//FUNCTION_BLOCK TcAxis_Tc2_MC2 EXTENDS TcAxis_Base IMPLEMENTS itfAxis_Tc2_MC2
//FUNCTION_BLOCK TcAxis_Tc2_MC2 EXTENDS TcAxis_DMC_Tc3_Direct_Motion_Control IMPLEMENTS itfAxis_Tc2_MC2
FUNCTION_BLOCK TcAxis_Tc2_MC2 IMPLEMENTS itfAxis_Tc2_MC2
//FUNCTION_BLOCK TcAxis_Tc2_MC2 EXTENDS TcAxis_Base IMPLEMENTS itfAxis_Tc3_DriveMotionControl, itfAxis_Tc2_MC2

//VAR_INPUT
//	Axis 				: Tc2_MC2.AXIS_REF;
//END_VAR
//VAR_OUTPUT
//END_VAR
VAR_IN_OUT 
	Axis 				: Tc2_MC2.AXIS_REF;
END_VAR
VAR	
	_PowerOn : BOOL;
//	itfCommand      : itfCommand;

//	_fbCommand       	: TcCommand;
	
	_fbAxisCommand   	: TcAxisCommand;

//itfAxisCommand  : itfAxisCommand;
//_Command         : ST_Command;
	

MC : ST_Tc2_MC2;	

count_delete : INT;	
END_VAR

 ACT_Cyclic_Update();

METHOD AbortTrigger : itfCommand
VAR_INPUT
END_VAR
END_METHOD

{warning 'add method implementation '}
METHOD AccelerationProfile 	: itfCommand
VAR_INPUT
	TimeScale				: REAL;
	AccelerationScale		: REAL;
	Offset					: REAL;
	BufferMode				: MC_BUFFER_MODE;
END_VAR
VAR
	
END_VAR
count_delete  := count_delete + 1;
END_METHOD

ACTION ACT_Cyclic_Update:
//update local variables from hardware
Axis.ReadStatus();
END_ACTION

{warning 'add property implementation'}
PROPERTY ActualPosition : REAL
GET
//Actual Position
IF Axis.Status.OpMode.Modulo THEN
    ActualPosition := Axis.NcToPlc.ModuloActPos;
ELSE
    ActualPosition := Axis.NcToPlc.ActPos;
END_IF

count_delete  := count_delete + 1;
END_GET
END_PROPERTY

{warning 'add property implementation'}
PROPERTY ActualTorque : REAL
GET
ActualTorque := Axis.NcToPlc.ActTorque;

count_delete  := count_delete + 1;
END_GET
END_PROPERTY

{warning 'add property implementation'}
PROPERTY ActualVelocity : REAL
GET
//Actual Velocity
ActualVelocity := Axis.NcToPlc.ActVelo;
END_GET
END_PROPERTY

{warning 'add property implementation'}
PROPERTY AxisWarning : BOOL
GET
count_delete  := count_delete + 1;
END_GET
END_PROPERTY

{warning 'add property implementation'}
PROPERTY CommunicationReady : BOOL
GET
count_delete  := count_delete + 1;
END_GET
END_PROPERTY

{warning 'add property implementation'}
PROPERTY Direction : AXIS_DIRECTION
GET
count_delete  := count_delete + 1;
END_GET
END_PROPERTY

PROPERTY Error : BOOL
GET
Error :=  Axis.Status.Error;
END_GET
END_PROPERTY

{warning 'add property implementation'}
PROPERTY ErrorId : WORD
GET

//ErrorId := Axis.Status.ErrorID;

count_delete  := count_delete + 1;
END_GET
END_PROPERTY

PROPERTY ErrorId_Udint_Status : UDINT
GET
ErrorId_Udint_Status := Axis.Status.ErrorID;
END_GET
END_PROPERTY

PROPERTY Geared : BOOL
GET
Geared :=  Axis.Status.Coupled;
//Axis.NcToPlc.CoupleState
END_GET
END_PROPERTY

{attribute 'TcRpcEnable'}
METHOD GearIn 			: itfSynchronizedAxisCommand
VAR_INPUT
	RatioNumerator		: LREAL;
	RatioDenominator	: UINT;
	Acceleration		: LREAL;
	Deceleration		: LREAL;
	Jerk				: LREAL;
//	BufferMode			: Tc2_MC2.MC_BufferMode; //Currently not implemented
//	Options             : Tc2_MC2.ST_GearInOptions; //Currently not implemented
END_VAR
VAR_IN_OUT 
	Slave				: Tc2_MC2.AXIS_REF;	
END_VAR
VAR
//	fbGearIn			: Tc2_MC2.MC_GearIn;	
END_VAR
	
MC.GearIn(
	Master:= Axis, 
	Slave:= Slave, 
	Execute:= TRUE, 
	RatioNumerator:= RatioNumerator, 
	RatioDenominator:= RatioDenominator, 
	Acceleration:= Acceleration,
	Deceleration:= Deceleration, 
	Jerk:= Jerk, 
	BufferMode:= , //BufferMode,
	Options:= , //Options, 
	InGear=> ,//Geared , 
	Busy=> , 
	Active=> , 
	CommandAborted=> , 
	Error=> , 
	ErrorID=> );
	
MC.GearIn(
	Master:= Axis, 
	Slave:= Slave, 
	Execute:= FALSE);
	
count_delete  := count_delete + 1;
END_METHOD

{attribute 'TcRpcEnable'}
METHOD GearInDyn 		: itfSynchronizedAxisCommand
VAR_INPUT
    GearRatio			: LREAL;
	Acceleration		: REAL;
	Deceleration		: REAL;
	Jerk				: REAL;
//	BufferMode			: Tc2_MC2.MC_BufferMode;
//	Options             : Tc2_MC2.ST_GearInDynOptions;
END_VAR

VAR_IN_OUT 
	Slave				: Tc2_MC2.AXIS_REF;	
END_VAR
END_METHOD

{attribute 'TcRpcEnable'}
METHOD GearInMultimaster 	: itfSynchronizedAxisCommand
VAR_INPUT
	GearRatio1				: LREAL;
	GearRatio2				: LREAL;
	GearRatio3				: LREAL;	
	GearRatio4				: LREAL;	
	Acceleration			: LREAL;
	Deceleration			: LREAL;
	Jerk					: LREAL;
	BufferMode				: Tc2_MC2.MC_BufferMode;
	Options             	: Tc2_MC2.ST_GearInMultiMasterOptions;	
END_VAR

VAR_IN_OUT
	Master1					: Tc2_MC2.AXIS_REF;	
	Master2					: Tc2_MC2.AXIS_REF;	
	Master3					: Tc2_MC2.AXIS_REF;	
	Master4					: Tc2_MC2.AXIS_REF;	
	Slave					: Tc2_MC2.AXIS_REF;	
END_VAR
END_METHOD

{attribute 'TcRpcEnable'}
METHOD GearOut 			: itfSynchronizedAxisCommand
VAR_INPUT
	Options             : Tc2_MC2.ST_GearInDynOptions;
END_VAR

VAR_IN_OUT 
	Slave				: Tc2_MC2.AXIS_REF;	
END_VAR
END_METHOD

{warning 'add method implementation '}
METHOD Halt 		: itfAxisCommand
VAR_INPUT
	Deceleration	: REAL;
	Jerk			: REAL;
	BufferMode		: MC_BUFFER_MODE;
END_VAR
VAR
//	fbHalt			: Tc2_MC2.MC_HALT;
END_VAR

MC.Halt(
	Axis:= Axis, 
	Execute:= , 
	Deceleration:= Deceleration, 
	Jerk:= Jerk, 
	BufferMode:= , //BufferMode, 
	Options:= , 
	Done=> , 
	Busy=> , 
	Active=> , 
	CommandAborted=> , 
	Error=> , 
	ErrorID=> );

count_delete  := count_delete + 1;
END_METHOD

{warning 'add method implementation '}
METHOD HaltSuperimposed : itfAxisCommand
VAR_INPUT
	Deceleration		: REAL;
	Jerk				: REAL;
END_VAR
VAR
	
END_VAR
count_delete  := count_delete + 1;
END_METHOD

{warning 'add method implementation '}
METHOD Home 		: itfAxisCommand
VAR_INPUT
	Position		: REAL;
	Velocity		: REAL;
	EndVelocity		: REAL;
	Acceleration	: REAL;
	Deceleration	: REAL;
	Jerk			: REAL;
	Direction		: MC_Direction;
	HomingMode		: INT;
	BufferMode		: MC_BUFFER_MODE;
END_VAR
VAR
//	fbHome			: Tc2_MC2.MC_HOME;
END_VAR

MC.Home(
	Axis:= Axis, 
	Execute:= TRUE, 
	Position:= Position, 
	HomingMode:= HomingMode, 
	BufferMode:= ,//BufferMode , 
	Options:= , 
	bCalibrationCam:= , 
	Done=> , 
	Busy=> , 
	Active=> , 
	CommandAborted=> , 
	Error=> , 
	ErrorID=> );

count_delete  := count_delete + 1;
END_METHOD

{warning 'add property implementation'}
PROPERTY HomeAbsSwitch : BOOL
GET
count_delete  := count_delete + 1;
END_GET
END_PROPERTY


PROPERTY IsHomed : BOOL
GET

IsHomed := Axis.Status.Homed;
END_GET
END_PROPERTY

{warning 'add method implementation '}
METHOD Jog 			: itfAxisCommand
VAR_INPUT
    JogForward 		: BOOL;
    JogBackwards 	: BOOL;
    Mode     		: Tc2_MC2.E_JogMode;
    Position        : LREAL;
    Velocity        : LREAL;
    Acceleration 	: LREAL;
    Deceleration 	: LREAL;
    Jerk     		: LREAL;
END_VAR
VAR
//	fbJog			: Tc2_MC2.MC_JOG;
END_VAR

MC.Jog(
	Axis:= Axis, 
	JogForward:= JogForward, 
	JogBackwards:= JogBackwards, 
	Mode:= Mode, 
	Position:= Position, 
	Velocity:= Velocity, 
	Acceleration:= Acceleration, 
	Deceleration:= Deceleration, 
	Jerk:= Jerk, 
	Done=> , 
	Busy=> , 
	Active=> , 
	CommandAborted=> , 
	Error=> , 
	ErrorID=> );


count_delete  := count_delete + 1;
END_METHOD

{warning 'add property implementation'}
PROPERTY LimitSwitchNegative : BOOL
GET

LimitSwitchNegative := Axis.Status.SoftLimitMinExceeded;

count_delete  := count_delete + 1;
END_GET
END_PROPERTY

{warning 'add property implementation'}
PROPERTY LimitSwitchPositive : BOOL
GET

LimitSwitchPositive := Axis.Status.SoftLimitMaxExceeded;

count_delete  := count_delete + 1;
END_GET
END_PROPERTY

{warning 'add property implementation'}
PROPERTY MotionStatus : MOTION_STATUS
GET
END_GET
END_PROPERTY

{attribute 'TcRpcEnable'}
METHOD MoveAbsolute : itfAxisCommand
VAR_INPUT
	Position		: REAL;
	Velocity		: REAL;
	Acceleration	: REAL;
	Deceleration	: REAL;
	Jerk			: REAL;
//	Direction		: MC_Direction;
	BufferMode		: MC_BUFFER_MODE;
//	Options         : Tc2_MC2.ST_MoveOptions;
	Options         : Tc2_Mc2.ST_MoveOptions;
END_VAR

VAR
	itfAxisCommand   : itfAxisCommand;
    _Command         : ST_Command;
END_VAR
itfAxisCommand := _fbAxisCommand;
	
MC.MoveAbsolute(
	Axis:= Axis, 
	Execute:= TRUE ,//Execute, //
	Position:= Position, 
	Velocity:= Velocity, 
	Acceleration:= Acceleration, 
	Deceleration:= Deceleration, 
	Jerk:= Jerk, 
	BufferMode:= BufferMode,//BufferMode, 
	Options:= Options, //Options, 
	Done=> _Command.Done, 
	Busy=> _Command.Busy, 
	Active=>_Command.Active, 
	CommandAborted=> _Command.CommandAborted, 
	Error=> _Command.Error, 
	ErrorID=> _Command.ErrorID_Udint);
	
MC.MoveAbsolute(
	Axis:= Axis, 
	Execute:= FALSE);	

itfAxisCommand.Done 				:=  _Command.Done AND ActualPosition = Position;             
itfAxisCommand.Busy   				:=	_Command.Busy;
itfAxisCommand.Active 				:=	_Command.Active;
itfAxisCommand.CommandAborted		:=	_Command.CommandAborted;
itfAxisCommand.Error 				:=	_Command.Error;
itfAxisCommand.ErrorID_Udint 		:=	_Command.ErrorID_Udint;

MoveAbsolute := itfAxisCommand;
END_METHOD

{warning 'add method implementation '}
METHOD MoveAdditive : itfAxisCommand
VAR_INPUT
	Distance		: REAL;
	Velocity		: REAL;
	Acceleration	: REAL;
	Deceleration	: REAL;
	Jerk			: REAL;
	BufferMode		: MC_BUFFER_MODE;
END_VAR
VAR
//	fbMoveAdditive 	: Tc2_MC2.MC_MoveAdditive;	
END_VAR

MC.MoveAdditive(
	Axis:= Axis, 
	Execute:= TRUE, 
	Distance:= Distance, 
	Velocity:= Velocity, 
	Acceleration:= Acceleration, 
	Deceleration:= Deceleration, 
	Jerk:= Jerk, 
	BufferMode:= , //BufferMode, 
	Options:= , 
	Done=> , 
	Busy=> , 
	Active=> , 
	CommandAborted=> , 
	Error=> , 
	ErrorID=> );


count_delete  := count_delete + 1;
END_METHOD

{warning 'add method implementation '}
METHOD MoveContinuousAbsolute 	: itfContinuousAxisCommand
VAR_INPUT
	Position					: REAL;
	EndVelocity					: REAL;
	Velocity					: REAL;
	Acceleration				: REAL;
	Deceleration				: REAL;
	Jerk						: REAL;
	Direction					: MC_DIRECTION;
	BufferMode					: MC_BUFFER_MODE;
END_VAR
VAR
//	fbMoveContinuousAbsolute 	: Tc2_MC2.MC_MoveContinuousAbsolute;		
END_VAR

MC.MoveContinuousAbsolute(
	Axis:= Axis, 
	Execute:= TRUE, 
	Position:= Position, 
	Velocity:= Velocity, 
	EndVelocity:= EndVelocity, 
	Acceleration:= Acceleration, 
	Deceleration:= Deceleration, 
	Jerk:= Jerk, 
	BufferMode:= ,//BufferMode, 
	Options:= , 
	InEndVelocity=> , 
	Busy=> , 
	Active=> , 
	CommandAborted=> , 
	Error=> , 
	ErrorID=> );


count_delete  := count_delete + 1;
END_METHOD

{warning 'add method implementation '}
METHOD MoveContinuousRelative 	: itfContinuousAxisCommand
VAR_INPUT
	Distance					: REAL;
	EndVelocity					: REAL;
	Velocity					: REAL;
	Acceleration				: REAL;
	Deceleration				: REAL;
	Jerk						: REAL;
	Direction					: MC_DIRECTION;
	BufferMode					: MC_BUFFER_MODE;
END_VAR
VAR
//	fbMoveContinuousRelative 	: Tc2_MC2.MC_MoveContinuousRelative;
END_VAR

MC.MoveContinuousRelative(
	Axis:= Axis, 
	Execute:= TRUE, 
	Distance:= Distance, 
	Velocity:= Velocity, 
	EndVelocity:= EndVelocity, 
	Acceleration:= Acceleration, 
	Deceleration:= Deceleration, 
	Jerk:= Jerk, 
	BufferMode:= ,//BufferMode, 
	Options:= , 
	InEndVelocity=> , 
	Busy=> , 
	Active=> , 
	CommandAborted=> , 
	Error=> , 
	ErrorID=> );



count_delete  := count_delete + 1;
END_METHOD

METHOD MoveModulo : itfAxisCommand
VAR_INPUT
END_VAR

MC.MoveModulo(
	Axis:= Axis, 
	Execute:= TRUE, 
	Position:= , 
	Velocity:= , 
	Acceleration:= , 
	Deceleration:= , 
	Jerk:= , 
	Direction:= , 
	BufferMode:= , 
	Options:= , 
	Done=> , 
	Busy=> , 
	Active=> , 
	CommandAborted=> , 
	Error=> , 
	ErrorID=> );
END_METHOD

{attribute 'TcRpcEnable'}
METHOD MoveRelative 	: itfAxisCommand
VAR_INPUT
	Distance			: REAL;
	Velocity			: REAL;
	Acceleration		: REAL;
	Deceleration		: REAL;
	Jerk				: REAL;
	BufferMode			: MC_BUFFER_MODE;
	Options         	: TC2_MC2.ST_MoveOptions;
END_VAR
VAR
	itfAxisCommand   : itfAxisCommand;
	_Command         : ST_Command;
END_VAR
itfAxisCommand := _fbAxisCommand;

MC.MoveRelative(
	Axis:= Axis, 
	Execute:= TRUE, 
	Distance:= Distance, 
	Velocity:= Velocity, 
	Acceleration:= Acceleration, 
	Deceleration:= Deceleration, 
	Jerk:= Jerk, 
	BufferMode:= ,//BufferMode, 
	Options:= Options, 
	Done=> _Command.Done, 
	Busy=> _Command.Busy, 
	Active=> _Command.Active, 
	CommandAborted=> _Command.CommandAborted, 
	Error=> _Command.Error, 
	ErrorID=> _Command.ErrorID_Udint);
	
MC.MoveRelative(
	Axis:= Axis, 
	Execute:= FALSE);		
	
itfAxisCommand.Done 				:=  _Command.Done; //AND ActualPosition = ActualPosition + Distance;             
itfAxisCommand.Busy   				:=	_Command.Busy;
itfAxisCommand.Active 				:=	_Command.Active;
itfAxisCommand.CommandAborted		:=	_Command.CommandAborted;
itfAxisCommand.Error 				:=	_Command.Error;
itfAxisCommand.ErrorID_Udint 		:=	_Command.ErrorID_Udint;

MoveRelative := itfAxisCommand;
END_METHOD

{warning 'add method implementation '}
METHOD MoveSuperimposed 	: itfAxisCommand
VAR_INPUT
	Distance				: REAL;
	VelocityDiff			: REAL;
	Acceleration			: REAL;
	Deceleration			: REAL;
	Jerk					: REAL;
END_VAR
VAR
//	fbMoveSuperimposed	 	: Tc2_MC2.MC_MoveSuperimposed;	
END_VAR

MC.MoveSuperimposed(
	Axis:= Axis, 
	Execute:= TRUE, 
	Mode:= , 
	Distance:= , 
	VelocityDiff:= VelocityDiff, 
	Acceleration:= Acceleration, 
	Deceleration:= Deceleration, 
	Jerk:= Jerk, 
	VelocityProcess:= , 
	Length:= , 
	Options:= , 
	Done=> , 
	Busy=> , 
	Active=> , 
	CommandAborted=> , 
	Error=> , 
	ErrorID=> , 
	Warning=> , 
	WarningId=> , 
	ActualVelocityDiff=> , 
	ActualDistance=> , 
	ActualLength=> , 
	ActualAcceleration=> , 
	ActualDeceleration=> );

count_delete  := count_delete + 1;
END_METHOD

{warning 'add method implementation '}
METHOD MoveVelocity 	: itfContinuousAxisCommand
VAR_INPUT
	Velocity			: REAL;
	Acceleration		: REAL;
	Deceleration		: REAL;
	Jerk				: REAL;
	Direction			: MC_Direction;
	BufferMode			: MC_BUFFER_MODE;
END_VAR
VAR
//	fbMoveVelocity	 	: Tc2_MC2.MC_MoveVelocity;	
END_VAR

MC.MoveVelocity(
	Axis:= Axis, 
	Execute:= TRUE, 
	Velocity:= Velocity, 
	Acceleration:= Acceleration, 
	Deceleration:= Deceleration, 
	Jerk:= Jerk, 
	Direction:= Direction, 
	BufferMode:= , //BufferMode
	Options:= , 
	InVelocity=> , 
	Busy=> , 
	Active=> , 
	CommandAborted=> , 
	Error=> , 
	ErrorID=> );	

count_delete  := count_delete + 1;
END_METHOD

{warning 'add method implementation '}
METHOD PhasingAbsolute 	: itfSynchronizedAxisCommand
VAR_INPUT
//	Master				: itfAxis;
	Master				: Tc2_MC2.AXIS_REF;
	Slave				: Tc2_MC2.AXIS_REF;		
	PhaseShift			: REAL;
	Velocity			: REAL;
	Acceleration		: REAL;
	Deceleration		: REAL;
	Jerk				: REAL;
	BufferMode			: MC_BUFFER_MODE;
END_VAR
VAR
//	fbPhasingAbsolute	: Tc2_MC2.MC_PhasingAbsolute;
END_VAR

MC.PhasingAbsolute(
	Master:= Master, 
	Slave:= Slave, 
	Execute:= TRUE, 
	ContinuousUpdate:= , 
	PhaseShift:= , 
	Velocity:= , 
	Acceleration:= , 
	Deceleration:= , 
	Jerk:= , 
	BufferMode:= , 
	Options:= , 
	Done=> , 
	Busy=> , 
	Active=> , 
	CommandAborted=> , 
	Error=> , 
	ErrorID=> , 
	AbsolutePhaseShift=> );

count_delete  := count_delete + 1;
END_METHOD

{warning 'add method implementation '}
METHOD PhasingRelative 	: itfSynchronizedAxisCommand
VAR_INPUT
//	Master				: itfAxis;
	Master				: Tc2_MC2.AXIS_REF;
	Slave				: Tc2_MC2.AXIS_REF;		
	PhaseShift			: REAL;
	Velocity			: REAL;
	Acceleration		: REAL;
	Deceleration		: REAL;
	Jerk				: REAL;
	BufferMode			: MC_BUFFER_MODE;
END_VAR
VAR
//	fbPhasingRelative	: Tc2_MC2.MC_PhasingRelative;
END_VAR

MC.PhasingRelative(
	Master:= Master, 
	Slave:= Slave, 
	Execute:= , 
	ContinuousUpdate:= , 
	PhaseShift:= , 
	Velocity:= , 
	Acceleration:= , 
	Deceleration:= , 
	Jerk:= , 
	BufferMode:= , 
	Options:= , 
	Done=> , 
	Busy=> , 
	Active=> , 
	CommandAborted=> , 
	Error=> , 
	ErrorID=> , 
	CoveredPhaseShift=> );

count_delete  := count_delete + 1;
END_METHOD

{warning 'add method implementation '}
METHOD PositionProfile 	: itfCommand
VAR_INPUT
	TimeScale			: REAL;
	PositionScale		: REAL;
	Offset				: REAL;
	BufferMode			: MC_BUFFER_MODE;
END_VAR
VAR
//	fbPositionProfile	 	: Tc2_MC2.;	
END_VAR






count_delete  := count_delete + 1;
END_METHOD

{attribute 'TcRpcEnable'}
METHOD Power 		: itfCommand
VAR_INPUT
	Enable			: BOOL;
	EnablePositive	: BOOL;
	EnableNegative	: BOOL;
END_VAR
VAR
	_fbCommand      : TcCommand;
	itfCommand      : itfCommand;
	Command         : ST_Command;
END_VAR

itfCommand := _fbCommand;

MC.Power(
	Axis:= Axis, 
	Enable:= Enable, 
	Enable_Positive:= EnablePositive, 
	Enable_Negative:= EnableNegative, 
	Override:= 100, 
	BufferMode:= , 
	Options:= , 
	Status=> Command.Status, 
	Busy=> Command.Busy,
	Active=> Command.Active,
	Error=> Command.Error,
	ErrorID=> Command.ErrorID_Udint);

itfCommand.Status		:=	Command.Status;
itfCommand.Busy   		:=	Command.Busy;
itfCommand.Active 		:=	Command.Active;
itfCommand.Error 		:=	Command.Error;
itfCommand.ErrorID_Udint :=	Command.ErrorID_Udint;
	
Power := itfCommand;

_PowerOn := MC.Power.Enable;
END_METHOD

{attribute ‘monitoring’ := ‘call’}
PROPERTY PowerOn : BOOL
GET
PowerOn := _PowerOn;
END_GET
END_PROPERTY

{warning 'add method implementation '}
METHOD ReadBoolParameter 	: MC_Error
VAR_INPUT
	ParameterNumber			: INT;
END_VAR
VAR_OUTPUT
	Value					: BOOL;
END_VAR
VAR
//	fbReadBoolParameter 	: Tc2_MC2.MC_ReadBoolParameter;
END_VAR

MC.ReadBoolParameter(
	Axis:= Axis, 
	Enable:= TRUE, 
	ParameterNumber:= ParameterNumber, 
	ReadMode:= , 
	Valid=> , 
	Busy=> , 
	Error=> , 
	ErrorID=> , 
	Value=> Value);


count_delete  := count_delete + 1;
END_METHOD

{warning 'add method implementation '}
METHOD ReadParameter 	: MC_Error
VAR_INPUT
	ParameterNumber		: INT;
END_VAR
VAR_OUTPUT
	Value				: REAL;
END_VAR
VAR
//	fbReadParameter		: Tc2_MC2.MC_ReadParameter;
END_VAR

MC.ReadParameter(
	Axis:= Axis, 
	Enable:= TRUE, 
	ParameterNumber:= ParameterNumber, 
	ReadMode:= , 
	Valid=> , 
	Busy=> , 
	Error=> , 
	ErrorID=> , 
	Value=> Value);


count_delete  := count_delete + 1;
END_METHOD

{warning 'add property implementation'}
PROPERTY ReadyForPowerOn : BOOL
GET
count_delete  := count_delete + 1;
END_GET
END_PROPERTY

{warning 'add method implementation '}
METHOD Release : MC_Error

VAR
	
END_VAR
count_delete  := count_delete + 1;
END_METHOD

{attribute 'TcRpcEnable'}
METHOD Reset 		: itfCommand

VAR
//	fbReset 		: Tc2_MC2.MC_RESET;
END_VAR

MC.Reset(
	Axis:= Axis, 
	Execute:= TRUE, 
	Done=> , 
	Busy=> , 
	Error=> , 
	ErrorID=> );


count_delete  := count_delete + 1;
END_METHOD

{warning 'add method implementation '}
METHOD SetOverride 	: MC_Error
VAR_INPUT
	VelFactor		: REAL;
	AccFactor		: REAL;
	JerkFactor		: REAL;
END_VAR

VAR
//	fbSetOverride 	: Tc2_MC2.MC_SetOverride;
END_VAR

MC.SetOverride(
	Axis:= Axis, 
	Enable:= TRUE, 
	VelFactor:= VelFactor, 
	AccFactor:= AccFactor, 
	JerkFactor:= JerkFactor, 
	Enabled=> , 
	Busy=> , 
	Error=> , 
	ErrorID=> );

count_delete  := count_delete + 1;
END_METHOD

{warning 'add method implementation '}
METHOD SetPosition 	: itfCommand
VAR_INPUT
	Position		: REAL;
	Relative		: BOOL; (* RELATIVE=True, ABSOLUTE=False (Default)*)
//	ExecutionMode	: MC_ExecutionMode;
    ExecutionMode	: Tc2_MC2.ST_SetPositionOptions;
END_VAR

VAR
//	fbSetPosition 	: Tc2_MC2.MC_SetPosition;
END_VAR

MC.SetPosition(
	Axis:= Axis, 
	Execute:= TRUE, 
	Position:= Position, 
	Mode:= Relative, 
	Options:= ExecutionMode, 
	Done=> , 
	Busy=> , 
	Error=> , 
	ErrorID=> );

count_delete  := count_delete + 1;
END_METHOD

{warning 'add property implementation'}
PROPERTY Simulation : BOOL
GET
count_delete  := count_delete + 1;
END_GET
END_PROPERTY

{attribute ‘monitoring’ := ‘call’}
PROPERTY Status : Tc2_MC2.MC_AxisStates
GET
VAR	
	AxisStates : Tc2_MC2.MC_AxisStates;
END_VAR

//CASE Axis.Status.MotionState OF 
//     MC_AXISSTATE_UNDEFINED : 
//         AxisStates := MC_AxisStates.MC_AXISSTATE_UNDEFINED;
//	MC_AXISSTATE_DISABLED:
//		AxisStates := MC_AxisStates.MC_AXISSTATE_DISABLED;
//	MC_AXISSTATE_STANDSTILL:
//		AxisStates := MC_AxisStates.MC_AXISSTATE_STANDSTILL;
//	MC_AXISSTATE_ERRORSTOP:		
//		AxisStates := MC_AxisStates.MC_AXISSTATE_ERRORSTOP;
//	MC_AXISSTATE_STOPPING:			
//		AxisStates := MC_AxisStates.MC_AXISSTATE_STOPPING;
//	MC_AXISSTATE_HOMING:			
//		AxisStates := MC_AxisStates.MC_AXISSTATE_HOMING;
//	MC_AXISSTATE_DISCRETEMOTION:			
//		AxisStates := MC_AxisStates.MC_AXISSTATE_DISCRETEMOTION;
//	MC_AXISSTATE_CONTINOUSMOTION:			
//		AxisStates := MC_AxisStates.MC_AXISSTATE_CONTINOUSMOTION;
//	MC_AXISSTATE_SYNCHRONIZEDMOTION:			
//		AxisStates := MC_AxisStates.MC_AXISSTATE_SYNCHRONIZEDMOTION;
//END_CASE;

//Status := AxisStates;

Status := Axis.Status.MotionState;
END_GET
END_PROPERTY

{warning 'add method implementation '}
METHOD Stop 		: itfAxisCommand
VAR_INPUT
	Deceleration	: REAL;
	Jerk			: REAL;
END_VAR
VAR
//	fbStop			: Tc2_MC2.MC_STOP;
END_VAR

MC.Stop(
	Axis:= Axis, 
	Execute:= TRUE, 
	Deceleration:= Deceleration, 
	Jerk:= Jerk, 
	Options:= , 
	Done=> , 
	Busy=> , 
	Active=> , 
	CommandAborted=> , 
	Error=> , 
	ErrorID=> );

count_delete  := count_delete + 1;
END_METHOD

{warning 'add method implementation '}
METHOD TorqueControl 	: itfAxisCommand
VAR_INPUT
	Torque				: REAL;
	TorqueRamp			: REAL;
	Velocity			: REAL;
	Acceleration		: REAL;
	Deceleration		: REAL;
	Jerk				: REAL;
	Direction			: MC_DIRECTION;
	BufferMode			: MC_BUFFER_MODE;
END_VAR
VAR
//	fbTorqueControl		: Tc2_MC2.MC_TorqueControl;
END_VAR

MC.TorqueControl(
	Axis:= Axis, 
	Execute:= , 
	ContinuousUpdate:= , 
	Relative:= , 
	Torque:= Torque, 
	TorqueRamp:= TorqueRamp, 
	VelocityLimitHigh:= , 
	VelocityLimitLow:= , 
	BufferMode:= , 
	Options:= , 
	InTorque=> , 
	Busy=> , 
	Active=> , 
	CommandAborted=> , 
	Error=> , 
	ErrorId=> );

count_delete  := count_delete + 1;
END_METHOD

METHOD TouchProbe : itfCommand
VAR_INPUT
END_VAR
END_METHOD

{warning 'add method implementation '}
METHOD VelocityProfile 	: itfCommand
VAR_INPUT
	TimeScale			: REAL;
	VelocityScale		: REAL;
	Offset				: REAL;
	BufferMode			: MC_BUFFER_MODE;
END_VAR
VAR
	
END_VAR
count_delete  := count_delete + 1;
END_METHOD

{warning 'add method implementation '}
METHOD WriteBoolParameter 	: MC_Error
VAR_INPUT
	ParameterNumber			: INT;
	Value					: BOOL;
END_VAR

VAR
//	fbWriteBoolParameter 	: Tc2_MC2.MC_WriteBoolParameter;	
END_VAR

MC.WriteBoolParameter(
	Axis:= Axis, 
	Execute:= TRUE, 
	ParameterNumber:= ParameterNumber, 
	Value:= Value, 
	Done=> , 
	Busy=> , 
	Error=> , 
	ErrorID=> );

count_delete  := count_delete + 1;
END_METHOD

{warning 'add method implementation '}
METHOD WriteParameter 	: MC_Error
VAR_INPUT
	ParameterNumber		: INT;
	Value				: REAL;
END_VAR

VAR
//	fbWriteParameter 	: Tc2_MC2.MC_WriteParameter;	
END_VAR

MC.WriteParameter(
	Axis:= Axis, 
	Execute:= TRUE, 
	ParameterNumber:= ParameterNumber, 
	Value:= Value, 
	Done=> , 
	Busy=> , 
	Error=> , 
	ErrorID=> );

count_delete  := count_delete + 1;
END_METHOD

END_FUNCTION_BLOCK

(* stored: Version 1.1.0.1, ProductVersion 3.1.4024.12
   POU TcAxis_Tc2_MC2: Id {ede46f14-de41-4cbf-bc63-b5cbbe198a41}, SpecialFunc None
   Folder ActualValues: Id {1a660d81-33e9-4cb9-b03a-13d277bb9b98}
   Folder Control: Id {1f231ae8-3c7d-437f-95f0-04b859b8036f}
   Folder MultiAxesMotion: Id {44c4f412-6645-404f-9d81-e01de0858822}
   Folder SingleAxisMotion: Id {773962eb-b74d-45a8-b24d-288626989ff0}
   Folder Status: Id {03058b18-c49a-4761-8ec3-e8bf4e5aa1d1}
   Folder Touch Probe: Id {a5f81912-eef1-4913-a787-44651389cb63}
   Method AbortTrigger: Id {7e7b714c-aa2c-4a74-95f0-6833e466216b}
   Method AccelerationProfile: Id {2d031de7-aa1e-4760-a585-3c08e8401237}
   Action ACT_Cyclic_Update: Id {5de5cd23-c71a-4817-8d0e-2b699f35e45d}
   Property ActualPosition: Id {b2230e07-cc2f-43f9-96fa-b3df5126c4b7}
   Get Get: Id {263c22f1-18b5-4f5f-aaf7-577af67fd31c}
   Property ActualTorque: Id {47f1f1a8-2481-48da-95ea-96476db64d77}
   Get Get: Id {d6e8535c-3af3-4c34-9d6d-c19c9f0a01f9}
   Property ActualVelocity: Id {e88b58fe-48b9-430f-bfde-dfb33c3bd932}
   Get Get: Id {7dc6c552-9454-4328-bbea-4a267ff83920}
   Property AxisWarning: Id {9681de72-c409-4b72-b04e-79507da56814}
   Get Get: Id {c6dd67f0-6fed-44ce-93f1-e538fdf76ea4}
   Property CommunicationReady: Id {8590d5ed-42e3-4ce6-b3e6-b01dc7d93a0c}
   Get Get: Id {02038667-914b-4c42-be19-d587813289b9}
   Property Direction: Id {aa7ab63a-8922-49c4-8310-24f5a4f0c70a}
   Get Get: Id {c552097b-2c34-4812-8ba6-f4c7cdf8fa48}
   Property Error: Id {73f39bd4-ba95-46df-a05d-3fbd114dc241}
   Get Get: Id {10691733-5fe1-4205-8dc2-ea19fc1c63cd}
   Property ErrorId: Id {f6537c7d-f19e-43d1-9730-38ba00377bec}
   Get Get: Id {3bd1eb7c-f586-4717-bdce-f7ce6a124431}
   Property ErrorId_Udint_Status: Id {d1af9492-b775-4c4c-9c2e-e16f7984c79e}
   Get Get: Id {b143cfd2-79d5-493b-8a6d-901da710f66c}
   Property Geared: Id {cad8364b-d06c-481a-9940-549f97d5ccbb}
   Get Get: Id {a3b3f0fb-2772-49f7-8dbb-75c9f3fa0511}
   Method GearIn: Id {6cbcc261-b3fb-4547-98ae-75e372afb64e}
   Method GearInDyn: Id {34f00123-93c7-4112-97a2-6bdb32b75f1f}
   Method GearInMultimaster: Id {e4118677-a979-4510-8b94-478ec510771a}
   Method GearOut: Id {b80af787-0897-496c-b2c3-680f811a2c90}
   Method Halt: Id {b5e61c76-4253-4650-9c4d-72d7a3b44126}
   Method HaltSuperimposed: Id {8e24962f-1f8b-45e3-9fd9-5cdc51b672a3}
   Method Home: Id {af023316-0daa-480a-9620-216f87d5a5f0}
   Property HomeAbsSwitch: Id {11667e14-831c-4aef-9a5a-39ccba0528ec}
   Get Get: Id {832ad001-4747-41e7-a8b4-939cb85c1540}
   Property IsHomed: Id {c73206de-8ef9-4ef0-a314-f9781e86939a}
   Get Get: Id {7ad0df17-5302-4856-973c-eae74fba749a}
   Method Jog: Id {b217b8a0-5ed3-4962-b3d8-ab876323bb77}
   Property LimitSwitchNegative: Id {07b013c4-fa8c-4e4e-b880-b99a700f2294}
   Get Get: Id {d7d494ad-a8d7-456e-bd2e-97fc8f5da81e}
   Property LimitSwitchPositive: Id {8f9e18ea-d405-4e05-86dd-8e0e6b996cd8}
   Get Get: Id {ed0f687e-30b9-4b4e-9a95-1745cbb04882}
   Property MotionStatus: Id {13fa6222-30dd-4861-963e-f23a6aee8455}
   Get Get: Id {0b5c4fb5-9547-4781-99c0-311b7cf4ea1e}
   Method MoveAbsolute: Id {75c5779f-04ff-4069-95d9-d7a1de4e344e}
   Method MoveAdditive: Id {41ab44ec-7746-4f1c-885f-94c8dd766d4e}
   Method MoveContinuousAbsolute: Id {33e3848e-94a8-499f-bd0e-8a5c066a1f3c}
   Method MoveContinuousRelative: Id {bcd4836b-509a-4705-81e4-3c0e0c808801}
   Method MoveModulo: Id {e498b0d0-5eab-4e87-b643-9fc1e9a96f1d}
   Method MoveRelative: Id {fddf74c6-fdb2-4e7c-a07f-3af72833d590}
   Method MoveSuperimposed: Id {64695090-d2ac-4903-bbe7-a60c98f2edf6}
   Method MoveVelocity: Id {c0d6a530-ab89-47b6-a229-25b41e577faa}
   Method PhasingAbsolute: Id {6636a02f-2e18-4d37-a884-ab23bb4c93d0}
   Method PhasingRelative: Id {7ec8289a-3b22-4471-a355-5030111af3bc}
   Method PositionProfile: Id {a2b258ae-89cc-4e69-a9bd-78deefeaefb9}
   Method Power: Id {f479a0c0-c959-4273-841a-a53ca6e59e8b}
   Property PowerOn: Id {788c8284-a067-4b73-bd3e-a5329fda0703}
   Get Get: Id {4debc66c-8c89-4b05-b196-32da99b6b0be}
   Method ReadBoolParameter: Id {fc75e571-fa59-4330-8562-ad247d6d290f}
   Method ReadParameter: Id {cddb6be3-68c2-4b4d-9c14-6a1de51eb2c5}
   Property ReadyForPowerOn: Id {7edfc666-a58e-4cdd-b6d9-ce309d3dbb55}
   Get Get: Id {5d7ca864-08a1-4fb9-b227-2975391c3e77}
   Method Release: Id {8b47a037-d6fc-4c76-8724-440d9cebf9dd}
   Method Reset: Id {14e50d85-e296-43cf-afd5-3cba42896a29}
   Method SetOverride: Id {159befbb-0e58-4754-96a4-765c9befbe12}
   Method SetPosition: Id {841fdfbb-6ac2-4c9c-b9c9-a0bf821b2be7}
   Property Simulation: Id {8db6e099-f6ba-4ea8-96dc-469ed58bba45}
   Get Get: Id {8573d2f0-d796-44a5-8d11-4f09bec709b2}
   Property Status: Id {899ae5c5-cb0d-4a4d-9f83-26636f1764e2}
   Get Get: Id {d011a0b2-92b3-4928-b561-f5a955384b13}
   Method Stop: Id {c7df0714-0c83-44e1-9182-81c8a840aa7d}
   Method TorqueControl: Id {6e3ef885-3d26-42b8-9949-5a5da1bc6ad2}
   Method TouchProbe: Id {9724a4d0-7f15-4489-9615-ca6b57fe446e}
   Method VelocityProfile: Id {ae47a6cf-f02b-4ff4-9871-0cd776202783}
   Method WriteBoolParameter: Id {3378c903-7622-4419-977d-9abca44ccb6f}
   Method WriteParameter: Id {45c39499-1570-46c6-aa44-5d04439c023a} *)
